{attribute 'qualified_only'}
{attribute 'strict'}
{attribute 'to_string'}
TYPE E_SeqDoors :
(
	IDLE := 0,
	
	//Outer door
	CLOSE_OUTER_DOOR,
	OUTER_DOOR_CLOSED,
	OPEN_OUTER_DOOR,
	OUTER_DOOR_OPENED,
		
	//Cleanroom door
	LOCK_CLEANROOM_DOOR,
	CLEANROOM_DOOR_LOCKED,
	RELEASE_CLEANROOM_DOOR,
	CLEANROOM_DOOR_RELEASED,
	
	READY := 10000,
	ERROR := 20000	
);
END_TYPE

(* stored: Version 1.1.0.1, ProductVersion 3.1.4024.12
   DUT E_SeqDoors: Id {dbd3de09-19ec-40e8-8b7c-04e0c63fda09} *)
